(* PLC project Unnamed, Unknown Unnamed 1 *)
(* stored: creationDateTime 2025-09-20T13:41:17, modificationDateTime 2025-09-24T22:36:35 *)

PROGRAM program0
  VAR_EXTERNAL
    X1 : BOOL;
    X2 : BOOL;
    Y1 : BOOL;
    Y2 : BOOL;
    Y3 : BOOL;
    Y4 : BOOL;
  END_VAR
  VAR
    cnt_rst : BOOL;
    run : BOOL := 0;
    blinker : BOOL := 0;
    tdelay : TIME := T#50ms;
    cnt_max : INT := 4;
    cnt_val : INT;
    const0 : INT := 0;
    const1 : INT := 1;
    const2 : INT := 2;
    const3 : INT := 3;
    TOF0 : TOF;
    TON0 : TON;
    CTU0 : CTU;
  END_VAR
  VAR  (* added by the conversion: wires and edge detectors of the diagram *)
    R_TRIG1 : R_TRIG;
  END_VAR

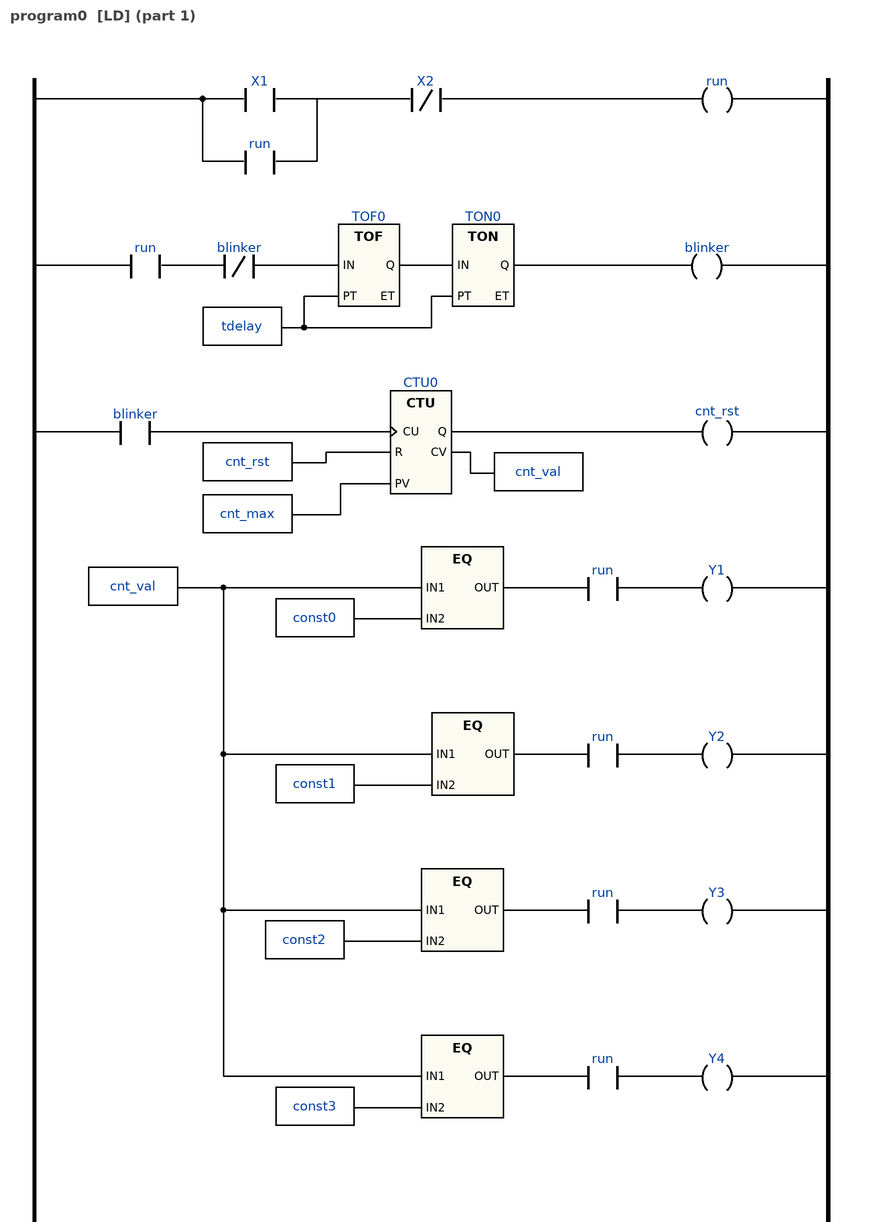
(* LD diagram, written out as Structured Text *)
run := (run OR X1) AND NOT X2;
R_TRIG1(CLK := blinker);
CTU0(CU := R_TRIG1.Q, R := cnt_rst, PV := cnt_max);
cnt_rst := CTU0.Q;
TOF0(IN := run AND NOT blinker, PT := tdelay);
TON0(IN := TOF0.Q, PT := tdelay);
blinker := TON0.Q;
cnt_val := CTU0.CV;
Y1 := cnt_val = const0 AND run;
Y2 := cnt_val = const1 AND run;
Y3 := cnt_val = const2 AND run;
Y4 := cnt_val = const3 AND run;
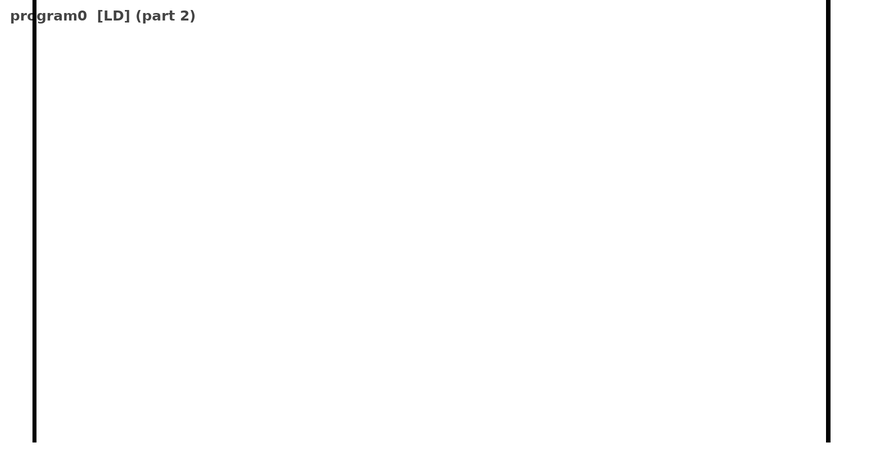
END_PROGRAM

CONFIGURATION config
  RESOURCE resource1 ON PLC
    VAR_GLOBAL
      X1 : BOOL;
      X2 : BOOL;
      X3 : BOOL;
      X4 : BOOL;
      Y1 : BOOL;
      Y2 : BOOL;
      Y3 : BOOL;
      Y4 : BOOL;
    END_VAR
    TASK task0(INTERVAL := T#25ms, PRIORITY := 0);
    PROGRAM instance0 WITH task0 : program0;
  END_RESOURCE
END_CONFIGURATION
